(* IEC 61131-3 sources: beckhoffAutomationInterface/ST/Shark/Lib/Subsystems, 8 files *)

(* ---- GVL_SubsystemSizes.st ---- *)
{attribute 'qualified_only'}
VAR_GLOBAL CONSTANT
    // FB_DoorLock: maximum proximity sensors per lock actuator.
    MAX_SENSORS_PER_LOCK      : INT := 4;

    // FB_DigitalInputSubsystem: maximum registered digital inputs.
    MAX_DIGITAL_INPUTS        : INT := 128;

    // FB_DigitalOutputSubsystem: maximum registered digital outputs.
    MAX_DIGITAL_OUTPUTS       : INT := 128;

    // FB_FlowSubsystem: maximum MFC zones.
    MAX_FLOW_ZONES            : INT := 64;

    // FB_PressureSubsystem: maximum pressure sensors.
    MAX_PRESSURE_SENSORS      : INT := 32;

    // FB_PressureSubsystem: maximum pressure controllers.
    MAX_PRESSURE_CONTROLLERS  : INT := 32;

    // FB_ValveSubsystem: maximum valve instances.
    MAX_VALVES                : INT := 256;
END_VAR

(* ---- FB_DigitalInputSubsystem.st ---- *)
// Lib digital-input subsystem.
//
// Owns a small fixed-capacity array of I_DigitalInput references. Count
// (and the array's effective range) is supplied by the caller at Init time
// via the App-side GVL constant. Lib code never references App enums or GVL.
FUNCTION_BLOCK FB_DigitalInputSubsystem IMPLEMENTS I_DigitalInputSubsystem
VAR_OUTPUT
    bInitialized : BOOL := FALSE;
END_VAR
VAR
    _aipInputs : ARRAY[1..GVL_SubsystemSizes.MAX_DIGITAL_INPUTS] OF I_DigitalInput;
    _nCount    : INT := 0;
END_VAR

METHOD PUBLIC Init : BOOL
VAR_INPUT
    aipInputs : ARRAY[*] OF I_DigitalInput;
    nCount    : INT;
END_VAR
VAR
    i      : INT;
    nLower : DINT;
END_VAR
    IF bInitialized THEN
        Init := TRUE;
        RETURN;
    END_IF

    IF nCount < 1 OR nCount > GVL_SubsystemSizes.MAX_DIGITAL_INPUTS THEN
        RETURN;
    END_IF

    nLower := LOWER_BOUND(aipInputs, 1);
    IF nCount > (UPPER_BOUND(aipInputs, 1) - nLower + 1) THEN
        RETURN;
    END_IF

    _nCount := nCount;
    FOR i := 1 TO _nCount DO
        _aipInputs[i] := aipInputs[nLower + i - 1];
    END_FOR

    bInitialized := TRUE;
    Init := TRUE;
END_METHOD

METHOD PUBLIC Execute : BOOL
    Execute := TRUE;
END_METHOD

METHOD PUBLIC IsInitialized : BOOL
    IsInitialized := bInitialized;
END_METHOD

METHOD PUBLIC GetCount : INT
    GetCount := _nCount;
END_METHOD

METHOD PUBLIC GetInputByIndex : I_DigitalInput
VAR_INPUT
    nInput : INT;
END_VAR
    IF nInput >= 1 AND nInput <= _nCount THEN
        GetInputByIndex := _aipInputs[nInput];
    ELSE
        GetInputByIndex := 0;
    END_IF
END_METHOD

METHOD PUBLIC GetStateByIndex : BOOL
VAR_INPUT
    nInput : INT;
END_VAR
VAR
    ipInput : I_DigitalInput;
END_VAR
    ipInput := GetInputByIndex(nInput);
    IF ipInput <> 0 THEN
        GetStateByIndex := ipInput.GetState();
    END_IF
END_METHOD

END_FUNCTION_BLOCK

(* ---- FB_DigitalOutputSubsystem.st ---- *)
// Lib digital-output subsystem.
//
// Owns a small fixed-capacity array of I_DigitalOutput references. Count
// (and the array's effective range) is supplied by the caller at Init time
// via the App-side GVL constant. Lib code never references App enums or GVL.
FUNCTION_BLOCK FB_DigitalOutputSubsystem IMPLEMENTS I_DigitalOutputSubsystem
VAR_OUTPUT
    bInitialized : BOOL := FALSE;
END_VAR
VAR
    _aipOutputs : ARRAY[1..GVL_SubsystemSizes.MAX_DIGITAL_OUTPUTS] OF I_DigitalOutput;
    _nCount     : INT := 0;
END_VAR

METHOD PUBLIC Init : BOOL
VAR_INPUT
    aipOutputs : ARRAY[*] OF I_DigitalOutput;
    nCount     : INT;
END_VAR
VAR
    i      : INT;
    nLower : DINT;
END_VAR
    IF bInitialized THEN
        Init := TRUE;
        RETURN;
    END_IF

    IF nCount < 1 OR nCount > GVL_SubsystemSizes.MAX_DIGITAL_OUTPUTS THEN
        RETURN;
    END_IF

    nLower := LOWER_BOUND(aipOutputs, 1);
    IF nCount > (UPPER_BOUND(aipOutputs, 1) - nLower + 1) THEN
        RETURN;
    END_IF

    _nCount := nCount;
    FOR i := 1 TO _nCount DO
        _aipOutputs[i] := aipOutputs[nLower + i - 1];
    END_FOR

    bInitialized := TRUE;
    Init := TRUE;
END_METHOD

METHOD PUBLIC Execute : BOOL
    Execute := TRUE;
END_METHOD

METHOD PUBLIC IsInitialized : BOOL
    IsInitialized := bInitialized;
END_METHOD

METHOD PUBLIC GetCount : INT
    GetCount := _nCount;
END_METHOD

METHOD PUBLIC GetOutputByIndex : I_DigitalOutput
VAR_INPUT
    nOutput : INT;
END_VAR
    IF nOutput >= 1 AND nOutput <= _nCount THEN
        GetOutputByIndex := _aipOutputs[nOutput];
    ELSE
        GetOutputByIndex := 0;
    END_IF
END_METHOD

METHOD PUBLIC SetOutputByIndex : BOOL
VAR_INPUT
    nOutput : INT;
    bValue  : BOOL;
END_VAR
VAR
    ipOutput : I_DigitalOutput;
END_VAR
    ipOutput := GetOutputByIndex(nOutput);
    IF ipOutput <> 0 THEN
        ipOutput.SetOutput(bValue);
        SetOutputByIndex := TRUE;
    END_IF
END_METHOD

METHOD PUBLIC GetStateByIndex : BOOL
VAR_INPUT
    nOutput : INT;
END_VAR
VAR
    ipOutput : I_DigitalOutput;
END_VAR
    ipOutput := GetOutputByIndex(nOutput);
    IF ipOutput <> 0 THEN
        GetStateByIndex := ipOutput.GetOutput();
    END_IF
END_METHOD

END_FUNCTION_BLOCK

(* ---- FB_DoorLock.st ---- *)
(*
FB_DoorLock — Controls a door lock output and aggregates its proximity sensors.

Composite pattern: a lock owns N FB_DoorSensor children (1..GVL_SubsystemSizes.MAX_SENSORS_PER_LOCK).
AllSensorsClosed iterates only sensors that were registered via AddSensor — a lock
with 1 sensor and a lock with 2 sensors both work correctly without any code change.
*)
FUNCTION_BLOCK FB_DoorLock
VAR
    _ipOutput     : I_DigitalOutput;
    _afbSensors   : ARRAY[1..GVL_SubsystemSizes.MAX_SENSORS_PER_LOCK] OF FB_DoorSensor;
    _nSensorCount : INT := 0;
    _bInitialized : BOOL := FALSE;
END_VAR

METHOD PUBLIC Init : BOOL
VAR_INPUT
    ipOutput : I_DigitalOutput;
END_VAR
    IF ipOutput = 0 THEN
        RETURN;
    END_IF
    _ipOutput     := ipOutput;
    _nSensorCount := 0;
    _bInitialized := TRUE;
    Init := TRUE;
END_METHOD

METHOD PUBLIC AddSensor : BOOL
VAR_INPUT
    ipInput : I_DigitalInput;
    bInvert : BOOL := FALSE;
END_VAR
    IF _nSensorCount >= GVL_SubsystemSizes.MAX_SENSORS_PER_LOCK THEN
        RETURN;
    END_IF
    IF _afbSensors[_nSensorCount + 1].Init(ipInput := ipInput, bInvert := bInvert) THEN
        _nSensorCount := _nSensorCount + 1;
        AddSensor := TRUE;
    END_IF
END_METHOD

METHOD PUBLIC Lock
    IF _bInitialized AND_THEN _ipOutput <> 0 THEN
        _ipOutput.SetOutput(TRUE);
    END_IF
END_METHOD

METHOD PUBLIC Unlock
    IF _bInitialized AND_THEN _ipOutput <> 0 THEN
        _ipOutput.SetOutput(FALSE);
    END_IF
END_METHOD

PROPERTY PUBLIC IsLocked : BOOL
    GET
        IF _bInitialized AND_THEN _ipOutput <> 0 THEN
            IsLocked := _ipOutput.GetOutput();
        END_IF
    END_GET
END_PROPERTY

METHOD PUBLIC AllSensorsClosed : BOOL
VAR
    i : INT;
END_VAR
    // Composite: iterate only registered sensors (not the full array bound)
    AllSensorsClosed := TRUE;
    FOR i := 1 TO _nSensorCount DO
        IF NOT _afbSensors[i].IsClosed THEN
            AllSensorsClosed := FALSE;
            RETURN;
        END_IF
    END_FOR
END_METHOD

END_FUNCTION_BLOCK

(* ---- FB_DoorSensor.st ---- *)
(*
FB_DoorSensor — Wraps an I_DigitalInput to represent a door proximity sensor.

Null Object pattern: an uninitialised sensor always reports IsClosed = FALSE
(door assumed open — the safe default for any safety or interlock logic).

bInvert: pass TRUE for normally-closed sensors where a LOW signal means closed.
*)
FUNCTION_BLOCK FB_DoorSensor
VAR
    _ipInput      : I_DigitalInput;
    _bInvert      : BOOL := FALSE;
    _bInitialized : BOOL := FALSE;
END_VAR

METHOD PUBLIC Init : BOOL
VAR_INPUT
    ipInput : I_DigitalInput;
    bInvert : BOOL := FALSE;
END_VAR
    IF ipInput = 0 THEN
        RETURN;
    END_IF
    _ipInput      := ipInput;
    _bInvert      := bInvert;
    _bInitialized := TRUE;
    Init := TRUE;
END_METHOD

PROPERTY PUBLIC IsClosed : BOOL
    GET
        // Null Object: uninitialized returns FALSE (door assumed open — safe default)
        IF _bInitialized AND_THEN _ipInput <> 0 THEN
            IsClosed := _ipInput.GetState() XOR _bInvert;
        END_IF
    END_GET
END_PROPERTY

END_FUNCTION_BLOCK

(* ---- FB_FlowSubsystem.st ---- *)
// Lib flow subsystem.
//
// Owns a small fixed-capacity array of I_Controller references (one per MFC
// zone). Count is supplied by the caller at Init time via the App-side GVL
// constant. Lib code never references App enums or GVL.
FUNCTION_BLOCK FB_FlowSubsystem IMPLEMENTS I_FlowSubsystem
VAR_OUTPUT
    bInitialized : BOOL := FALSE;
    bAnyError    : BOOL := FALSE;
    stFirstError : ST_Error;
END_VAR
VAR
    _ipControllers : ARRAY[1..GVL_SubsystemSizes.MAX_FLOW_ZONES] OF I_Controller;
    _nCount        : INT := 0;
END_VAR

METHOD PUBLIC Init : BOOL
VAR_INPUT
    aipControllers : ARRAY[*] OF I_Controller;
    nCount         : INT;
END_VAR
VAR
    i      : INT;
    nLower : DINT;
END_VAR
    IF bInitialized THEN
        Init := TRUE;
        RETURN;
    END_IF

    IF nCount < 1 OR nCount > GVL_SubsystemSizes.MAX_FLOW_ZONES THEN
        RETURN;
    END_IF

    nLower := LOWER_BOUND(aipControllers, 1);
    IF nCount > (UPPER_BOUND(aipControllers, 1) - nLower + 1) THEN
        RETURN;
    END_IF

    _nCount := nCount;
    FOR i := 1 TO _nCount DO
        _ipControllers[i] := aipControllers[nLower + i - 1];
    END_FOR

    bInitialized := TRUE;
    Init := TRUE;
END_METHOD

METHOD PUBLIC Execute : BOOL
VAR
    i        : INT;
    stStatus : ST_ControllerStatus;
END_VAR
    bAnyError := FALSE;
    stFirstError.eErrorId := E_ErrorId.NO_ERROR;
    stFirstError.sSource := '';
    stFirstError.sMessage := '';

    FOR i := 1 TO _nCount DO
        IF _ipControllers[i] <> 0 THEN
            stStatus := _ipControllers[i].GetStatus();
            _CaptureFirstError(stStatus.stError);
        END_IF
    END_FOR

    Execute := TRUE;
END_METHOD

METHOD PRIVATE _CaptureFirstError
VAR_INPUT
    stError : ST_Error;
END_VAR
    IF stError.eErrorId <> E_ErrorId.NO_ERROR THEN
        bAnyError := TRUE;
        IF stFirstError.eErrorId = E_ErrorId.NO_ERROR THEN
            stFirstError := stError;
        END_IF
    END_IF
END_METHOD

METHOD PUBLIC IsInitialized : BOOL
    IsInitialized := bInitialized;
END_METHOD

METHOD PUBLIC HasAnyError : BOOL
    HasAnyError := bAnyError;
END_METHOD

METHOD PUBLIC GetCount : INT
    GetCount := _nCount;
END_METHOD

METHOD PUBLIC GetControllerByIndex : I_Controller
VAR_INPUT
    nZone : INT;
END_VAR
    IF nZone >= 1 AND nZone <= _nCount THEN
        GetControllerByIndex := _ipControllers[nZone];
    ELSE
        GetControllerByIndex := 0;
    END_IF
END_METHOD

METHOD PUBLIC GetSensorByIndex : I_Sensor
VAR_INPUT
    nZone : INT;
END_VAR
VAR
    ipSensor : I_Sensor;
END_VAR
    IF nZone >= 1 AND nZone <= _nCount THEN
        IF _ipControllers[nZone] <> 0 AND_THEN __QUERYINTERFACE(_ipControllers[nZone], ipSensor) THEN
            GetSensorByIndex := ipSensor;
        END_IF
    END_IF
END_METHOD

END_FUNCTION_BLOCK

(* ---- FB_PressureSubsystem.st ---- *)
// Lib pressure subsystem.
//
// Owns two fixed-capacity arrays — pressure sensors and pressure controllers.
// Counts are supplied by the caller at Init time via App-side GVL constants.
// Lib code never references App enums or GVL.
FUNCTION_BLOCK FB_PressureSubsystem IMPLEMENTS I_PressureSubsystem
VAR_OUTPUT
    bInitialized : BOOL := FALSE;
    bAnyError    : BOOL := FALSE;
    stFirstError : ST_Error;
END_VAR
VAR
    _ipSensors        : ARRAY[1..GVL_SubsystemSizes.MAX_PRESSURE_SENSORS] OF I_Sensor;
    _ipControllers    : ARRAY[1..GVL_SubsystemSizes.MAX_PRESSURE_CONTROLLERS] OF I_Controller;
    _nSensorCount     : INT := 0;
    _nControllerCount : INT := 0;
END_VAR

METHOD PUBLIC Init : BOOL
VAR_INPUT
    aipSensors        : ARRAY[*] OF I_Sensor;
    nSensorCount      : INT;
    aipControllers    : ARRAY[*] OF I_Controller;
    nControllerCount  : INT;
END_VAR
VAR
    i        : INT;
    nLowerS  : DINT;
    nLowerC  : DINT;
END_VAR
    IF bInitialized THEN
        Init := TRUE;
        RETURN;
    END_IF

    IF nSensorCount < 0 OR nSensorCount > GVL_SubsystemSizes.MAX_PRESSURE_SENSORS THEN
        RETURN;
    END_IF
    IF nControllerCount < 0 OR nControllerCount > GVL_SubsystemSizes.MAX_PRESSURE_CONTROLLERS THEN
        RETURN;
    END_IF

    nLowerS := LOWER_BOUND(aipSensors, 1);
    IF nSensorCount > (UPPER_BOUND(aipSensors, 1) - nLowerS + 1) THEN
        RETURN;
    END_IF

    nLowerC := LOWER_BOUND(aipControllers, 1);
    IF nControllerCount > (UPPER_BOUND(aipControllers, 1) - nLowerC + 1) THEN
        RETURN;
    END_IF

    _nSensorCount := nSensorCount;
    FOR i := 1 TO _nSensorCount DO
        _ipSensors[i] := aipSensors[nLowerS + i - 1];
    END_FOR

    _nControllerCount := nControllerCount;
    FOR i := 1 TO _nControllerCount DO
        _ipControllers[i] := aipControllers[nLowerC + i - 1];
    END_FOR

    bInitialized := TRUE;
    Init := TRUE;
END_METHOD

METHOD PUBLIC Execute : BOOL
VAR
    i        : INT;
    stStatus : ST_ControllerStatus;
END_VAR
    bAnyError := FALSE;
    stFirstError.eErrorId := E_ErrorId.NO_ERROR;
    stFirstError.sSource := '';
    stFirstError.sMessage := '';

    FOR i := 1 TO _nSensorCount DO
        IF _ipSensors[i] <> 0 AND_THEN _ipSensors[i].IsError() THEN
            _CaptureFirstError(_ipSensors[i].GetError());
        END_IF
    END_FOR

    FOR i := 1 TO _nControllerCount DO
        IF _ipControllers[i] <> 0 THEN
            stStatus := _ipControllers[i].GetStatus();
            _CaptureFirstError(stStatus.stError);
        END_IF
    END_FOR

    Execute := TRUE;
END_METHOD

METHOD PRIVATE _CaptureFirstError
VAR_INPUT
    stError : ST_Error;
END_VAR
    IF stError.eErrorId <> E_ErrorId.NO_ERROR THEN
        bAnyError := TRUE;
        IF stFirstError.eErrorId = E_ErrorId.NO_ERROR THEN
            stFirstError := stError;
        END_IF
    END_IF
END_METHOD

METHOD PUBLIC IsInitialized : BOOL
    IsInitialized := bInitialized;
END_METHOD

METHOD PUBLIC HasAnyError : BOOL
    HasAnyError := bAnyError;
END_METHOD

METHOD PUBLIC GetSensorByIndex : I_Sensor
VAR_INPUT
    nSensor : INT;
END_VAR
    IF nSensor >= 1 AND nSensor <= _nSensorCount THEN
        GetSensorByIndex := _ipSensors[nSensor];
    ELSE
        GetSensorByIndex := 0;
    END_IF
END_METHOD

METHOD PUBLIC GetSensorCount : INT
    GetSensorCount := _nSensorCount;
END_METHOD

METHOD PUBLIC GetControllerByIndex : I_Controller
VAR_INPUT
    nCtrl : INT;
END_VAR
    IF nCtrl >= 1 AND nCtrl <= _nControllerCount THEN
        GetControllerByIndex := _ipControllers[nCtrl];
    ELSE
        GetControllerByIndex := 0;
    END_IF
END_METHOD

METHOD PUBLIC GetControllerCount : INT
    GetControllerCount := _nControllerCount;
END_METHOD

METHOD PUBLIC GetControllerAsSensorByIndex : I_Sensor
VAR_INPUT
    nCtrl : INT;
END_VAR
VAR
    ipSensor : I_Sensor;
END_VAR
    IF nCtrl >= 1 AND nCtrl <= _nControllerCount THEN
        IF _ipControllers[nCtrl] <> 0 AND_THEN __QUERYINTERFACE(_ipControllers[nCtrl], ipSensor) THEN
            GetControllerAsSensorByIndex := ipSensor;
        END_IF
    END_IF
END_METHOD

END_FUNCTION_BLOCK

(* ---- FB_ValveSubsystem.st ---- *)
// Lib valve subsystem.
//
// Owns a small fixed-capacity array of I_Valve references. Count is supplied
// by the caller at Init time via the App-side GVL constant. Lib code never
// references App enums or GVL.
FUNCTION_BLOCK FB_ValveSubsystem IMPLEMENTS I_ValveSubsystem
VAR_OUTPUT
    bInitialized : BOOL := FALSE;
    bAnyError    : BOOL := FALSE;
    stFirstError : ST_Error;
END_VAR
VAR
    _ipValves : ARRAY[1..GVL_SubsystemSizes.MAX_VALVES] OF I_Valve;
    _nCount   : INT := 0;
END_VAR

METHOD PUBLIC Init : BOOL
VAR_INPUT
    aipValves : ARRAY[*] OF I_Valve;
    nCount    : INT;
END_VAR
VAR
    i        : INT;
    nLower   : DINT;
END_VAR
    IF bInitialized THEN
        Init := TRUE;
        RETURN;
    END_IF

    IF nCount < 1 OR nCount > GVL_SubsystemSizes.MAX_VALVES THEN
        RETURN;
    END_IF

    nLower := LOWER_BOUND(aipValves, 1);
    IF nCount > (UPPER_BOUND(aipValves, 1) - nLower + 1) THEN
        RETURN;
    END_IF

    _nCount := nCount;
    FOR i := 1 TO _nCount DO
        _ipValves[i] := aipValves[nLower + i - 1];
    END_FOR

    bInitialized := TRUE;
    Init := TRUE;
END_METHOD

METHOD PUBLIC Execute : BOOL
VAR
    i : INT;
END_VAR
    bAnyError := FALSE;
    stFirstError.eErrorId := E_ErrorId.NO_ERROR;
    stFirstError.sSource  := '';
    stFirstError.sMessage := '';

    FOR i := 1 TO _nCount DO
        IF _ipValves[i] <> 0 AND_THEN _ipValves[i].IsError() THEN
            bAnyError := TRUE;
            IF stFirstError.eErrorId = E_ErrorId.NO_ERROR THEN
                stFirstError := _ipValves[i].GetError();
            END_IF
        END_IF
    END_FOR

    Execute := TRUE;
END_METHOD

METHOD PUBLIC IsInitialized : BOOL
    IsInitialized := bInitialized;
END_METHOD

METHOD PUBLIC HasAnyError : BOOL
    HasAnyError := bAnyError;
END_METHOD

METHOD PUBLIC GetValveByIndex : I_Valve
VAR_INPUT
    nValveId : INT;
END_VAR
    IF nValveId >= 1 AND nValveId <= _nCount THEN
        GetValveByIndex := _ipValves[nValveId];
    ELSE
        GetValveByIndex := 0;
    END_IF
END_METHOD

END_FUNCTION_BLOCK
